FUNCTION_BLOCK ListOfTest EXTENDS List
VAR_INPUT
END_VAR
VAR_OUTPUT
END_VAR
VAR
END_VAR

END_FUNCTION_BLOCK

(* stored: Version 1.1.0.1, ProductVersion 3.1.4024.11
   POU ListOfTest: Id {183e14cd-ee8b-4013-8501-80cf739dd2df}, SpecialFunc None *)
